TYPE DUT_PositionState :
// Include io: input on things that should never be mutable in EPICS.
// Omit io on things that may or may not need to be mutable, allow engineer to decide in their pragma.
// Currently: some installations would want position and delta to be mutable.
STRUCT
	{attribute 'pytmc' := '
		pv: NAME
		io: input
	'}
	sName: STRING;

	{attribute 'pytmc' := '
		pv: SETPOINT
	'}
	fPosition: LREAL;
	
	{attribute 'pytmc' := '
		pv: DELTA
	'}
	fDelta: LREAL;
	
	{attribute 'pytmc' := '
		pv: VELO
		io: input
	'}
	fVelocity: LREAL;
	
	{attribute 'pytmc' := '
		pv: ACCL
		io: input
	'}
	fAccel: LREAL;
	
	{attribute 'pytmc' := '
		pv: DCCL
		io: input
	'}
	fDecel: LREAL;
	
	{attribute 'pytmc' := '
		pv: VALID
		io: input
	'}
	bValid: BOOL := FALSE;
END_STRUCT
END_TYPE

(* stored: Version 1.1.0.1, ProductVersion 3.1.4022.12
   DUT DUT_PositionState: Id {85d45494-8a84-426c-8efe-9136ee5821c6} *)
